FUNCTION FC_Check_STX : BOOL
VAR_INPUT
	I_sString : REFERENCE TO T_MaxString;
END_VAR
VAR
	stringPos	: INT;
END_VAR

stringPos := FIND(I_sString, STX);
IF stringPos <> 0 THEN
	I_sString := MID(I_sString, LEN(I_sString), stringPos+1);
	FC_Check_STX := TRUE;
ELSE
	FC_Check_STX := FALSE;
END_IF

END_FUNCTION

(* stored: Version 1.1.0.1, ProductVersion 3.1.4024.15
   POU FC_Check_STX: Id {d2baa182-4a59-49a8-951e-920f00dd15ad}, SpecialFunc None *)
